// Mitsubishi GX Works2 project: MyProject-PLC   PLC: FX3U/FX3UC

PROGRAM MAIN
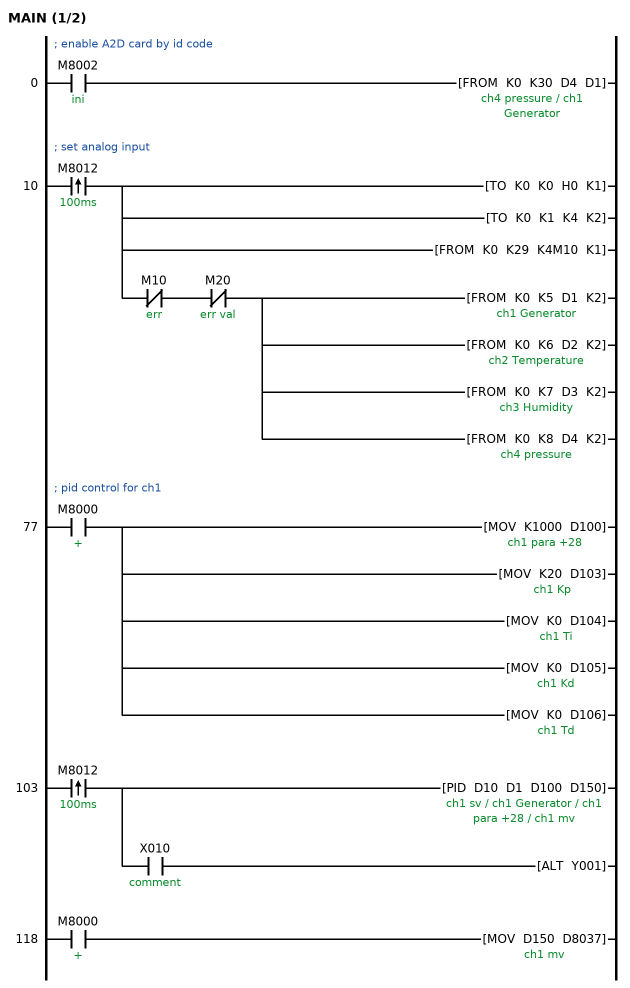
; enable A2D card by id code
0     LD      M8002  ; ini
      FROM    K0 K30 D4 D1  ; ch4 pressure / ch1 Generator
; set analog input
10    LDP     M8012  ; 100ms
      TO      K0 K0 H0 K1
      TO      K0 K1 K4 K2
      FROM    K0 K29 K4M10 K1  ; err
      ANI     M10  ; err
      ANI     M20  ; err val
      FROM    K0 K5 D1 K2
      FROM    K0 K6 D2 K2  ; ch2 Temperature
      FROM    K0 K7 D3 K2  ; ch3 Humidity
      FROM    K0 K8 D4 K2
; pid control for ch1
77    LD      M8000  ; +
      MOV     K1000 D100  ; ch1 para +28
      MOV     K20 D103  ; ch1 Kp
      MOV     K0 D104  ; ch1 Ti
      MOV     K0 D105  ; ch1 Kd
      MOV     K0 D106  ; ch1 Td
103   LDP     M8012  ; 100ms
      PID     D10 D1 D100 D150  ; ch1 sv / ch1 mv
      AND     X010  ; comment
      ALT     Y001
118   LD      M8000  ; +
      MOV     D150 D8037
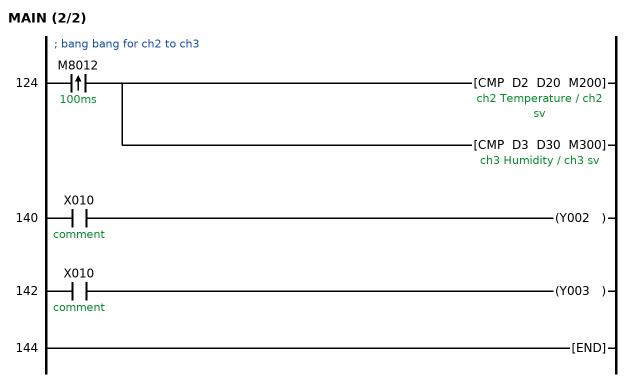
; bang bang for ch2 to ch3
124   LDP     M8012  ; 100ms
      CMP     D2 D20 M200  ; ch2 sv
      CMP     D3 D30 M300  ; ch3 sv
140   LD      X010  ; comment
      OUT     Y002
142   LD      X010  ; comment
      OUT     Y003
144   END
END_PROGRAM
